FUNCTION_BLOCK FB_LogToFile EXTENDS FB_CyclicFB

VAR CONSTANT
	LOG_SETTINGS 				: ST_LoggerSettings := (netID := '', filePath := 'C:\Logs\', filePrefix := 'SystemApp_', FileType := '.txt');	
	LOG_TIMEOUT 				: TIME := T#5S;
	EXPORT_INTERVAL				: TIME := T#10S;
	NEW_LINE 					: STRING(2) := '$r$n'; // Newline character
END_VAR

VAR
    ringBuffer 					: FB_StringRingBuffer;
    bufferMemory 				: ARRAY[0..5000] OF BYTE; // Adjust size as needed
	
	firstCycle 					: BOOL := TRUE;
	exportTimer					: TON;
	
	// From FB_init
    _netId 	 					: T_AmsNetId;     // Net ID for file operations
    _dirPath 					: T_MaxString;    // Directory path for the log file
	_logPrefix  				: STRING(10);     // Prefix for log file
	_fileExtension 				: STRING(10);  // File extension i.e. '.txt'
	_timeOut 					: TIME := DEFAULT_ADS_TIMEOUT;

// Params
	_execute 					: BOOL := FALSE; // Trigger for the log operation
    _data 	 					: T_MaxString; // Log entry to write

// Internal
	state 						: E_LogToFile_State;

    fileOpen  					: FB_FileOpen;
    fileClose 					: FB_FileClose;
    fileWrite 					: FB_FileWrite;

	fileRef 					: UINT := 0;       	// File handle
    risingEdge 					: R_TRIG;     // Rising edge detector for execute signal
END_VAR

VAR_OUTPUT
	smDone, smBusy, smError : BOOL;
    errId : UDINT;	 // Error ID in case of failure
END_VAR

METHOD CyclicLogic
VAR
	bufferFillPercentage: UDINT;
END_VAR
IF ( firstCycle ) THEN
	ringBuffer( pBuffer := ADR(bufferMemory), cbBuffer := SIZEOF(bufferMemory), bOverwrite := TRUE );
	firstCycle := FALSE;
	state := E_LogToFile_State.IDLE;
	RETURN;
END_IF

ringBuffer();

exportTimer(IN := TRUE, PT := EXPORT_INTERVAL);
bufferFillPercentage := (ringBuffer.cbSize * 100) / SIZEOF(bufferMemory);

IF ( ( exportTimer.Q  ) AND ( ringBuffer.nCount > 0 ) ) OR (bufferFillPercentage > 50) THEN
	//M_WriteToFile(); // Export logs when conditions are met
	_execute := TRUE;
	exportTimer(IN := FALSE); // Reset timer
ELSE
	_execute := FALSE;
END_IF;

M_StateMachine();
END_METHOD

//FB_Init is always available implicitly and it is used primarily for initialization.
//The return value is not evaluated. For a specific influence, you can also declare the
//methods explicitly and provide additional code there with the standard initialization
//code. You can evaluate the return value.
METHOD FB_Init: BOOL
VAR_INPUT
    bInitRetains: BOOL; // TRUE: the retain variables are initialized (reset warm / reset cold)
    bInCopyCode: BOOL;  // TRUE: the instance will be copied to the copy code afterward (online change)
END_VAR
_netID := LOG_SETTINGS.netID;
_dirPath := LOG_SETTINGS.filePath;
_logPrefix := LOG_SETTINGS.filePrefix;
_fileExtension := LOG_SETTINGS.FileType;
_timeOut := LOG_TIMEOUT;
END_METHOD

METHOD PUBLIC M_AddSysLog : BOOL

VAR_INPUT
    severity : INT;
    message : STRING;
END_VAR

VAR
    logEntry : STRING;
END_VAR
// Concatenate severity and message
logEntry := CONCAT('Severity ', INT_TO_STRING(severity));
logEntry := CONCAT(logEntry, ': ');
logEntry := CONCAT(logEntry, message);

// Add log entry to ring buffer
ringBuffer.A_AddTail(putValue := logEntry);
IF ( NOT ringbuffer.bOk ) THEN
	// Handle write error (optional)END_IF;
END_IF
END_METHOD

METHOD PRIVATE M_CloseFile : BOOL

VAR_INPUT
	execute : BOOL;	
END_VAR
IF ( NOT execute ) THEN
	fileOpen(bExecute := FALSE);
	M_CloseFile := FALSE;
	RETURN;
END_IF

IF ( NOT fileOpen.bBusy ) THEN     
	fileClose(sNetId := _netId, hFile := fileRef, tTimeout := _timeOut);
END_IF

// Attempt to close the file
fileClose(bExecute := TRUE);

IF ( NOT M_HandleError(fileClose.bError , fileClose.nErrId) ) THEN
	fileRef := 0; // File handle
END_IF

M_CloseFile := fileClose.bBusy;
END_METHOD

METHOD PRIVATE M_HandleError : BOOL
VAR_INPUT
	check 					: BOOL;
	errorID 				: UDINT;
END_VAR
check := error;

IF check THEN
	errId := errorID;
END_IF

M_HandleError := check;
END_METHOD

METHOD PRIVATE M_OpenFile : BOOL

VAR_INPUT
	execute 				: BOOL;	
END_VAR

VAR
	getSystemTime 			: GETSYSTEMTIME; // System time function block
	fileTime 				: T_FILETIME;     // File time
	dateString 				: STRING;		// Date string for filename
	filePath 				: STRING; 	// Full log file path
END_VAR
IF ( NOT execute ) THEN
	fileOpen(bExecute := FALSE);
	M_OpenFile := FALSE;
	RETURN;
END_IF

IF ( _dirPath = '' ) THEN
   	M_HandleError(TRUE , 99);
	M_OpenFile := FALSE;
    RETURN;
END_IF

IF ( NOT fileOpen.bBusy ) THEN
	// Generate log file path with current date
	getSystemTime(timeLoDW => fileTime.dwLowDateTime, timeHiDW => fileTime.dwHighDateTime );
	dateString := SYSTEMTIME_TO_STRING(FILETIME_TO_SYSTEMTIME(fileTime));
	filepath := CONCAT(_dirPath, _logPrefix); 			// Create file path
	filePath := CONCAT(filepath, LEFT(dateString, 10)); // Add date to file path
	filePath := CONCAT(filepath, _fileExtension); 		// Add file extension to file path.
     
	fileOpen(sNetId := '', sPathName := filePath, nMode := FOPEN_MODEAPPEND, ePath := PATH_GENERIC, tTimeout := _timeOut);
END_IF

// Attempt to open the file
fileOpen(bExecute := TRUE);

IF ( NOT M_HandleError(fileOpen.bError , fileOpen.nErrId) ) THEN
	fileRef := fileOpen.hFile; // No error case
END_IF

M_OpenFile := fileOpen.bBusy;
END_METHOD

METHOD M_StateMachine

VAR
	status			: BOOL;
END_VAR
RisingEdge(CLK := _execute);

CASE state OF
    E_LogToFile_State.IDLE: // Idle state
        IF ( RisingEdge.Q ) THEN
			smDone := FALSE;
           	smBusy := TRUE;
            smError := FALSE;
            errId := 0;
		
			fileOpen(bExecute := FALSE);
			fileWrite(bExecute := FALSE);
			fileClose(bExecute := FALSE);

            state := E_LogToFile_State.OPEN_FILE;
        END_IF

    E_LogToFile_State.OPEN_FILE: // Open the file
        status := M_OpenFile(TRUE);
		IF error THEN
			state := E_LogToFile_State.CLOSE_FILE;
        ELSIF ( fileRef <> 0 ) AND ( NOT status ) THEN
			M_OpenFile(FALSE);
			state := E_LogToFile_State.PREPARE_DATA;
        END_IF
		
	E_LogToFile_State.PREPARE_DATA:
		ringBuffer.A_RemoveHead();
		_data := ringBuffer.getValue;
		
		IF ( _data <> '' ) THEN
			M_WriteToFile(FALSE, '');
			state := E_LogToFile_State.WRITE_TO_FILE;
		ELSE
			IF ( NOT fileWrite.bBusy ) THEN
				state := E_LogToFile_State.CLOSE_FILE;
			END_IF
		END_IF
		
    E_LogToFile_State.WRITE_TO_FILE: // Write to the file
		status := M_WriteToFile(execute := TRUE, inputString := _data);
		
		IF ( NOT status ) THEN
			state := E_LogToFile_State.PREPARE_DATA;
		END_IF
	
    
    E_LogToFile_State.CLOSE_FILE: // Close the file
       IF ( fileREF <> 0 ) THEN
			status :=  M_CloseFile(TRUE);
			IF ( error OR ( NOT fileWrite.bBusy ) ) THEN
				M_CloseFile(FALSE);
				state := E_LogToFile_State.RESET;
        	END_IF
		ELSE
			M_CloseFile(FALSE);
			state := E_LogToFile_State.RESET;
	   END_IF

    E_LogToFile_State.RESET: // Cleanup and reset
		smDone := TRUE;
		smBusy := FALSE;
        fileRef := 0;;
        state := E_LogToFile_State.IDLE; // Return to idle state
END_CASE
END_METHOD

METHOD PRIVATE M_WriteToFile : BOOL

VAR_INPUT
	execute : BOOL;
	inputString : STRING; // Log entry to write
END_VAR

VAR
	msgString : STRING;
END_VAR
IF ( NOT execute ) THEN
	fileOpen(bExecute := FALSE);
	fileWrite(bExecute := FALSE);
	M_WriteToFile := FALSE;
	RETURN;
END_IF

IF ( NOT fileWrite.bBusy ) THEN
	
	IF ( LEN(inputString) > (UINT_TO_INT(SIZEOF(msgString)) - LEN(NEW_LINE))) THEN
		M_HandleError( TRUE, 98);
		M_WriteToFile := FALSE;
		RETURN;
	END_IF

	msgString := CONCAT( inputString, NEW_LINE );

	// Write the message to the file
	fileWrite(sNetId := _netId, hFile := fileRef, pWriteBuff := ADR(msgString), cbWriteLen := INT_TO_UDINT(LEN(msgString)), tTimeout := +_timeOut);
END_IF

// Attempt to write the file
fileWrite(bExecute := TRUE);

IF ( M_HandleError(fileWrite.bError , fileWrite.nErrId) ) THEN
	M_WriteToFile := FALSE; // File handle
	RETURN;
END_IF

M_WriteToFile := fileWrite.bBusy;
END_METHOD

END_FUNCTION_BLOCK

(* stored: Version 1.1.0.1
   POU FB_LogToFile: Id {fb5295cb-b1f0-49d5-9615-1a2a01ed1744}, SpecialFunc None
   Folder I_CyclicLogic: Id {87daa978-67c6-4a39-86ac-3d294411fb43}
   Folder Private: Id {fc975c30-933a-4e62-908f-c6744c85109e}
   Method CyclicLogic: Id {927c198c-b88a-4c95-956a-748cb57237df}
   Method FB_init: Id {9777b847-b97e-4dff-ae75-c6e3eaac3d98}
   Method M_AddSysLog: Id {1b2fb357-e815-4ace-afb2-8f3df1c1dad2}
   Method M_CloseFile: Id {d38a4b35-b3a5-43ee-bd0d-254ea85cb7ec}
   Method M_HandleError: Id {78e24d16-4370-48ca-b07a-c9807c919296}
   Method M_OpenFile: Id {265e6e42-3b42-4497-9b62-d63a0adb2967}
   Method M_StateMachine: Id {2fa36e72-1bf8-451a-8c2e-ff84f03be0d5}
   Method M_WriteToFile: Id {647db4ea-59c0-40ef-8b79-062cf0a303c0} *)
